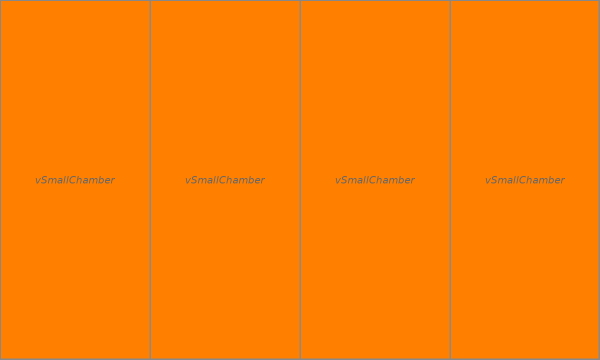
VISUALIZATION vStatusScreen  // 600x360
VAR_IN_OUT
	arChamber : 	ARRAY[0..3] OF fbChamber;
	arParams :   ARRAY[0..3] OF stParamsChamber;
	arControl :   ARRAY[0..3] OF stControl;
END_VAR
    Frame (0,0 150x360)
        shows vSmallChamber(stParams := arParams[0], fbChamber := arChamber[0], stControl := arControl[0])
    Frame (150,0 150x360)
        shows vSmallChamber(stParams := arParams[1], fbChamber := arChamber[1], stControl := arControl[1])
    Frame (450,0 150x360)
        shows vSmallChamber(stParams := arParams[3], fbChamber := arChamber[3], stControl := arControl[3])
    Frame (300,0 150x360)
        shows vSmallChamber(stParams := arParams[2], fbChamber := arChamber[2], stControl := arControl[2])
END_VISUALIZATION

(* stored: Version 1.1.0.1, ProductVersion 3.1.4024.12
   Visu vStatusScreen: Id {443c9623-b99a-4d49-ab5f-23885c3bde25} *)
